FUNCTION_BLOCK FB_TimeElapsed_HMI
VAR_INPUT
	i_RectWidth				:INT;
	i_tTimeActual			:TIME;
	i_tTimeSet				:TIME;
END_VAR
VAR_OUTPUT
	q_iValue				:REAL;
END_VAR
VAR
	iTimeActual_Min				:DINT;
	iTimeSet_Min				:DINT;
	fbScale						:FB_Scale;
END_VAR

iTimeSet_Min:=TIME_TO_DINT(i_tTimeSet)/100;
iTimeActual_Min:=TIME_TO_DINT(i_tTimeActual)/100;

IF iTimeSet_Min <> 0 THEN
	fbSCale(i_iValue:=DINT_TO_INT(iTimeActual_Min),
			i_iRawData_Low:=0,
			i_iRawData_High:=DINT_TO_INT(iTimeSet_Min),
			i_rScaled_Low:=0,
			i_rScaled_High:=i_RectWidth,
			i_rOffset:=0,
			q_rScaled=>q_iValue);
END_IF

END_FUNCTION_BLOCK

(* stored: Version 1.1.0.1, ProductVersion 3.1.4024.12
   POU FB_TimeElapsed_HMI: Id {d3c9f531-d565-421c-9b84-27919f12ef36}, SpecialFunc None *)
